FUNCTION_BLOCK INTERNAL FB_StringBuilderEx_Any_Tests EXTENDS TcUnit.FB_TestSuite
VAR_INPUT
END_VAR
VAR_OUTPUT
END_VAR
VAR
	stringBuilder	: FB_StringBuilder;
END_VAR

Test01_BOOL();
Test02_BYTE();
Test03_DATE();
Test04_DateAndTime();
Test05_DINT();
Test06_DWORD();
Test07_ENUM();
Test08_INT();
Test09_LINT();
Test10_LREAL();
Test11_LTIME();
Test12_LWORD();
Test13_REAL();
Test14_SINT();
Test15_STRING();
Test16_TIME();
Test17_TOD();
Test18_UDINT();
Test19_UINT();
Test20_ULINT();
Test21_USINT();
Test22_WORD();
Test23_WSTRING();
Test24_ANY_BIT_WORD();
Test25_ANY_BIT_BYTE();
Test26_ANY_BIT_DWORD();
Test27_ANY_BIT_LWORD();
Test28_ANY_REAL_REAL();
Test29_ANY_REAL_LREAL();

METHOD Test01_BOOL
VAR_INPUT
END_VAR

VAR_INST
	bTrue		: BOOL := TRUE;
	bFalse		: BOOL := FALSE;

END_VAR
IF TcUnit.TEST_ORDERED('Test01_BOOL') THEN
	AssertEquals_STRING(
		Actual := stringBuilder.Reset().AddAny(bTrue).Create(),
		Expected := 'TRUE',
		Message := 'Adding boolean failed');
		
	AssertEquals_STRING(
		Actual := stringBuilder.Reset().AddAny(bFalse).Create(),
		Expected := 'FALSE',
		Message := 'Adding boolean failed');
		
	TcUnit.TEST_FINISHED();
END_IF
END_METHOD

METHOD Test02_BYTE
VAR_INPUT
END_VAR
VAR
	byteVar	: BYTE := 17;
END_VAR
IF TEST_ORDERED('Test02_BYTE') THEN
	
	AssertEquals_STRING(
		Actual := stringBuilder.Reset().AddAny(byteVar).Create(),
		Expected := '17',
		Message := 'Adding BYTE failed.');
	TEST_FINISHED();
END_IF
END_METHOD

METHOD Test03_DATE
VAR
	someVar	: DATE := D#1970-01-01;
END_VAR
IF TEST_ORDERED('Test03_DATE') THEN
	AssertEquals_STRING(
		Actual := stringBuilder.Reset().AddAny(someVar).Create(),
		Expected := 'D#1970-01-01',
		Message := 'Adding DATE failed.');

	TEST_FINISHED();
END_IF
END_METHOD

METHOD Test04_DateAndTime
VAR
	someVar	: DATE_AND_TIME := DT#1970-1-1-0:0:1;
END_VAR
IF TEST_ORDERED('Test04_DateAndTime') THEN
	AssertEquals_STRING(
		Actual := stringBuilder.Reset().AddAny(someVar).Create(),
		Expected := 'DT#1970-01-01-00:00:01',
		Message := 'Adding DATE_AND_TIME failed.');

	TEST_FINISHED();
END_IF
END_METHOD

METHOD Test05_DINT
VAR
	someVar	: DINT := 15;
END_VAR
IF TEST_ORDERED('Test05_DINT') THEN
	AssertEquals_STRING(
		Actual := stringBuilder.Reset().AddAny(someVar).Create(),
		Expected := '15',
		Message := 'Adding DINT failed.');

	TEST_FINISHED();
END_IF
END_METHOD

METHOD Test06_DWORD
VAR
	someVar	: DWORD := 777;
END_VAR
IF TEST_ORDERED('Test06_DWORD') THEN
	AssertEquals_STRING(
		Actual := stringBuilder.Reset().AddAny(someVar).Create(),
		Expected := '777',
		Message := 'Adding DWORD failed.');

	TEST_FINISHED();
END_IF
END_METHOD

METHOD Test07_ENUM
VAR
	someVar	: E_AddAnyBitOptions := E_AddAnyBitOptions.HEXADECIMAL;
END_VAR
IF TEST_ORDERED('Test07_ENUM') THEN
	AssertEquals_STRING(
		Actual := stringBuilder.Reset().AddAny(someVar).Create(),
		Expected := '2',
		Message := 'Adding ENUM failed.');

	TEST_FINISHED();
END_IF
END_METHOD

METHOD Test08_INT
VAR
	someVar	: INT := 22;
END_VAR
IF TEST_ORDERED('Test08_INT') THEN
	AssertEquals_STRING(
		Actual := stringBuilder.Reset().AddAny(someVar).Create(),
		Expected := '22',
		Message := 'Adding INT failed.');

	TEST_FINISHED();
END_IF
END_METHOD

METHOD Test09_LINT
VAR
	someVar	: LINT := 6666;
END_VAR
IF TEST_ORDERED('Test09_LINT') THEN
	AssertEquals_STRING(
		Actual := stringBuilder.Reset().AddAny(someVar).Create(),
		Expected := '6666',
		Message := 'Adding LINT failed.');

	TEST_FINISHED();
END_IF
END_METHOD

METHOD Test10_LREAL
VAR
	someVar	: LREAL := 11.11;
END_VAR
IF TEST_ORDERED('Test10_LREAL') THEN
	AssertEquals_STRING(
		Actual := stringBuilder.Reset().AddAny(someVar).Create(),
		Expected := '11.11',
		Message := 'Adding LREAL failed.');

	TEST_FINISHED();
END_IF
END_METHOD

METHOD Test11_LTIME
VAR
	someVar	: LTIME := LTIME#100D2H30M40S500MS600US700NS;
END_VAR
IF TEST_ORDERED('Test11_LTIME') THEN
	AssertEquals_STRING(
		Actual := stringBuilder.Reset().AddAny(someVar).Create(),
		Expected := 'LTIME#100d2h30m40s500ms600us700ns',
		Message := 'Adding LTIME failed.');

	TEST_FINISHED();
END_IF
END_METHOD

METHOD Test12_LWORD
VAR
	someVar	: LWORD := 123456;
END_VAR
IF TEST_ORDERED('Test12_LWORD') THEN
	AssertEquals_STRING(
		Actual := stringBuilder.Reset().AddAny(someVar).Create(),
		Expected := '123456',
		Message := 'Adding LWORD failed.');

	TEST_FINISHED();
END_IF
END_METHOD

METHOD Test13_REAL
VAR
	someVar	: REAL := 12345.6789;
END_VAR
IF TEST_ORDERED('Test13_REAL') THEN
	AssertEquals_STRING(
		Actual := stringBuilder.Reset().AddAny(someVar).Create(),
		Expected := '12345.679',
		Message := 'Adding REAL failed.');

	TEST_FINISHED();
END_IF
END_METHOD

METHOD Test14_SINT
VAR
	someVar	: SINT := -34;
END_VAR
IF TEST_ORDERED('Test14_SINT') THEN
	AssertEquals_STRING(
		Actual := stringBuilder.Reset().AddAny(someVar).Create(),
		Expected := '-34',
		Message := 'Adding SINT failed.');

	TEST_FINISHED();
END_IF
END_METHOD

METHOD Test15_STRING
VAR
	someVar	: STRING := 'haha';
END_VAR
IF TEST_ORDERED('Test15_STRING') THEN
	AssertEquals_STRING(
		Actual := stringBuilder.Reset().AddAny(someVar).Create(),
		Expected := 'haha',
		Message := 'Adding STRING failed.');

	TEST_FINISHED();
END_IF
END_METHOD

METHOD Test16_TIME
VAR
	someVar	: TIME := T#15D10S;
END_VAR
IF TEST_ORDERED('Test16_TIME') THEN
	AssertEquals_STRING(
		Actual := stringBuilder.Reset().AddAny(someVar).Create(),
		Expected := 'T#15d10s',
		Message := 'Adding TIME failed.');

	TEST_FINISHED();
END_IF
END_METHOD

METHOD Test17_TOD
VAR
	someVar	: TOD := TOD#14:01:05.123;
END_VAR
IF TEST_ORDERED('Test17_TOD') THEN
	AssertEquals_STRING(
		Actual := stringBuilder.Reset().AddAny(someVar).Create(),
		Expected := 'TOD#14:01:05.123',
		Message := 'Adding TOD failed.');

	TEST_FINISHED();
END_IF
END_METHOD

METHOD Test18_UDINT
VAR
	someVar	: UDINT := 23452352;
END_VAR
IF TEST_ORDERED('Test18_UDINT') THEN
	AssertEquals_STRING(
		Actual := stringBuilder.Reset().AddAny(someVar).Create(),
		Expected := '23452352',
		Message := 'Adding UDINT failed.');

	TEST_FINISHED();
END_IF
END_METHOD

METHOD Test19_UINT
VAR
	someVar	: UINT := 12341;
END_VAR
IF TEST_ORDERED('Test19_UINT') THEN
	AssertEquals_STRING(
		Actual := stringBuilder.Reset().AddAny(someVar).Create(),
		Expected := '12341',
		Message := 'Adding UINT failed.');

	TEST_FINISHED();
END_IF
END_METHOD

METHOD Test20_ULINT
VAR
	someVar	: ULINT := 12345678;
END_VAR
IF TEST_ORDERED('Test20_ULINT') THEN
	AssertEquals_STRING(
		Actual := stringBuilder.Reset().AddAny(someVar).Create(),
		Expected := '12345678',
		Message := 'Adding ULINT failed.');

	TEST_FINISHED();
END_IF
END_METHOD

METHOD Test21_USINT
VAR
	someVar	: USINT := 123;
END_VAR
IF TEST_ORDERED('Test21_USINT') THEN
	AssertEquals_STRING(
		Actual := stringBuilder.Reset().AddAny(someVar).Create(),
		Expected := '123',
		Message := 'Adding USINT failed.');

	TEST_FINISHED();
END_IF
END_METHOD

METHOD Test22_WORD
VAR
	someVar	: WORD := 16#A;
END_VAR
IF TEST_ORDERED('Test22_WORD') THEN
	AssertEquals_STRING(
		Actual := stringBuilder.Reset().AddAny(someVar).Create(),
		Expected := '10',
		Message := 'Adding WORD failed.');

	TEST_FINISHED();
END_IF
END_METHOD

METHOD Test23_WSTRING
VAR
	someVar	: WSTRING := "test";
END_VAR
IF TEST_ORDERED('Test23_WSTRING') THEN
	AssertEquals_STRING(
		Actual := stringBuilder.Reset().AddAny(someVar).Create(),
		Expected := 'test',
		Message := 'Adding WSTRING failed.');

	TEST_FINISHED();
END_IF
END_METHOD

METHOD Test24_ANY_BIT_WORD
VAR_INPUT
END_VAR
VAR
	wordVar	: WORD := 16#AB;
	result	: Tc2_System.T_MaxString;
END_VAR
IF TcUnit.TEST_ORDERED('Test24_ANY_BIT_WORD') THEN
	
	// BINARY with notations
	result := stringBuilder.Reset().
		AddAnyBit(
			anyBit := wordVar, 
			option := E_AddAnyBitOptions.BINARY, 
			lowerCase := FALSE, 
			displayedDigitsCount := 16, 
			addNotation := TRUE)
		.Create();
		
	AssertEquals_STRING(
		Actual := result,
		Expected := '(BIN)0000000010101011',
		Message := 'Adding word as BINARY with addNotation = TRUE was incorrect');
		
	// BINARY without notations
	result := stringBuilder.Reset()
		.AddAnyBit(
			anyBit := wordVar, 
			option := E_AddAnyBitOptions.BINARY, 
			lowerCase := FALSE, 
			displayedDigitsCount := 16, 
			addNotation := FALSE)
		.Create();
		
	AssertEquals_STRING(
		Actual := result,
		Expected := '0000000010101011',
		Message := 'Adding word as BINARY with addNotation = FALSE was incorrect');
		
	// DECIMAL with notations
	result := stringBuilder.Reset()
		.AddAnyBit(
			anyBit := wordVar, 
			option := E_AddAnyBitOptions.DECIMAL, 
			lowerCase := FALSE, 
			displayedDigitsCount := 16, 
			addNotation := TRUE)
		.Create();
		
	AssertEquals_STRING(
		Actual := result,
		Expected := '(DEC)0000000000000171',
		Message := 'Adding word as DECIMAL with addNotation = TRUE was incorrect');
		
	// DECIMAL without notations
	result := stringBuilder.Reset()
		.AddAnyBit(
			anyBit := wordVar, 
			option := E_AddAnyBitOptions.DECIMAL, 
			lowerCase := FALSE, 
			displayedDigitsCount := 16, 
			addNotation := FALSE)
		.Create();
		
	AssertEquals_STRING(
		Actual := result,
		Expected := '0000000000000171',
		Message := 'Adding word as DECIMAL with addNotation = FALSE was incorrect');

	// HEXADECIMAL with notations
	result := stringBuilder.Reset()
		.AddAnyBit(
			anyBit := wordVar, 
			option := E_AddAnyBitOptions.HEXADECIMAL, 
			lowerCase := FALSE, 
			displayedDigitsCount := 16, 
			addNotation := TRUE)
		.Create();
		
	AssertEquals_STRING(
		Actual := result,
		Expected := '(HEX)00000000000000AB',
		Message := 'Adding word as HEXADECIMAL with addNotation = TRUE was incorrect');
		
	// HEXADECIMAL without notations
	result := stringBuilder.Reset()
		.AddAnyBit(
			anyBit := wordVar, 
			option := E_AddAnyBitOptions.HEXADECIMAL, 
			lowerCase := FALSE, 
			displayedDigitsCount := 16, 
			addNotation := FALSE)
		.Create();
		
	AssertEquals_STRING(
		Actual := result,
		Expected := '00000000000000AB',
		Message := 'Adding word as HEXADECIMAL with addNotation = FALSE was incorrect');
	
	// OCTAL with notations
	result := stringBuilder.Reset()
		.AddAnyBit(
			anyBit := wordVar, 
			option := E_AddAnyBitOptions.OCTAL, 
			lowerCase := FALSE, 
			displayedDigitsCount := 16, 
			addNotation := TRUE)
		.Create();
		
	AssertEquals_STRING(
		Actual := result,
		Expected := '(OCT)0000000000000253',
		Message := 'Adding word as OCTAL with addNotation = TRUE was incorrect');
		
	// OCTAL without notations
	result := stringBuilder.Reset()
		.AddAnyBit(
			anyBit := wordVar, 
			option := E_AddAnyBitOptions.OCTAL, 
			lowerCase := FALSE, 
			displayedDigitsCount := 16, 
			addNotation := FALSE)
		.Create();
		
	AssertEquals_STRING(
		Actual := result,
		Expected := '0000000000000253',
		Message := 'Adding word as OCTAL with addNotation = FALSE was incorrect');
		
	TcUnit.TEST_FINISHED();
END_IF
END_METHOD

METHOD Test25_ANY_BIT_BYTE
VAR_INPUT
END_VAR
VAR
	byteVar	: BYTE := 16#AB;
	result	: Tc2_System.T_MaxString;
END_VAR
IF TcUnit.TEST_ORDERED('Test25_ANY_BIT_BYTE') THEN
	
	// BINARY with notations
	result := stringBuilder.Reset().
		AddAnyBit(
			anyBit := byteVar, 
			option := E_AddAnyBitOptions.BINARY, 
			lowerCase := FALSE, 
			displayedDigitsCount := 8, 
			addNotation := TRUE)
		.Create();
		
	AssertEquals_STRING(
		Actual := result,
		Expected := '(BIN)10101011',
		Message := 'Adding byte as BINARY with addNotation = TRUE was incorrect');
		
	// BINARY without notations
	result := stringBuilder.Reset()
		.AddAnyBit(
			anyBit := byteVar, 
			option := E_AddAnyBitOptions.BINARY, 
			lowerCase := FALSE, 
			displayedDigitsCount := 8, 
			addNotation := FALSE)
		.Create();
		
	AssertEquals_STRING(
		Actual := result,
		Expected := '10101011',
		Message := 'Adding byte as BINARY with addNotation = FALSE was incorrect');
		
	// DECIMAL with notations
	result := stringBuilder.Reset()
		.AddAnyBit(
			anyBit := byteVar, 
			option := E_AddAnyBitOptions.DECIMAL, 
			lowerCase := FALSE, 
			displayedDigitsCount := 8, 
			addNotation := TRUE)
		.Create();
		
	AssertEquals_STRING(
		Actual := result,
		Expected := '(DEC)00000171',
		Message := 'Adding byte as DECIMAL with addNotation = TRUE was incorrect');
		
	// DECIMAL without notations
	result := stringBuilder.Reset()
		.AddAnyBit(
			anyBit := byteVar, 
			option := E_AddAnyBitOptions.DECIMAL, 
			lowerCase := FALSE, 
			displayedDigitsCount := 8, 
			addNotation := FALSE)
		.Create();
		
	AssertEquals_STRING(
		Actual := result,
		Expected := '00000171',
		Message := 'Adding byte as DECIMAL with addNotation = FALSE was incorrect');

	// HEXADECIMAL with notations
	result := stringBuilder.Reset()
		.AddAnyBit(
			anyBit := byteVar, 
			option := E_AddAnyBitOptions.HEXADECIMAL, 
			lowerCase := FALSE, 
			displayedDigitsCount := 8, 
			addNotation := TRUE)
		.Create();
		
	AssertEquals_STRING(
		Actual := result,
		Expected := '(HEX)000000AB',
		Message := 'Adding byte as HEXADECIMAL with addNotation = TRUE was incorrect');
		
	// HEXADECIMAL without notations
	result := stringBuilder.Reset()
		.AddAnyBit(
			anyBit := byteVar, 
			option := E_AddAnyBitOptions.HEXADECIMAL, 
			lowerCase := FALSE, 
			displayedDigitsCount := 8, 
			addNotation := FALSE)
		.Create();
		
	AssertEquals_STRING(
		Actual := result,
		Expected := '000000AB',
		Message := 'Adding byte as HEXADECIMAL with addNotation = FALSE was incorrect');
	
	// OCTAL with notations
	result := stringBuilder.Reset()
		.AddAnyBit(
			anyBit := byteVar, 
			option := E_AddAnyBitOptions.OCTAL, 
			lowerCase := FALSE, 
			displayedDigitsCount := 8, 
			addNotation := TRUE)
		.Create();
		
	AssertEquals_STRING(
		Actual := result,
		Expected := '(OCT)00000253',
		Message := 'Adding byte as OCTAL with addNotation = TRUE was incorrect');
		
	// OCTAL without notations
	result := stringBuilder.Reset()
		.AddAnyBit(
			anyBit := byteVar, 
			option := E_AddAnyBitOptions.OCTAL, 
			lowerCase := FALSE, 
			displayedDigitsCount := 8, 
			addNotation := FALSE)
		.Create();
		
	AssertEquals_STRING(
		Actual := result,
		Expected := '00000253',
		Message := 'Adding byte as OCTAL with addNotation = FALSE was incorrect');
		
	TcUnit.TEST_FINISHED();
END_IF
END_METHOD

METHOD Test26_ANY_BIT_DWORD
VAR
	dwordVar	: DWORD := 16#AB;
	result	: Tc2_System.T_MaxString;
END_VAR
IF TcUnit.TEST_ORDERED('Test26_ANY_BIT_DWORD') THEN
	
	// BINARY with notations
	result := stringBuilder.Reset().
		AddAnyBit(
			anyBit := dwordVar, 
			option := E_AddAnyBitOptions.BINARY, 
			lowerCase := FALSE, 
			displayedDigitsCount := 32, 
			addNotation := TRUE)
		.Create();
		
	AssertEquals_STRING(
		Actual := result,
		Expected := '(BIN)00000000000000000000000010101011',
		Message := 'Adding dword as BINARY with addNotation = TRUE was incorrect');
		
	// BINARY without notations
	result := stringBuilder.Reset()
		.AddAnyBit(
			anyBit := dwordVar, 
			option := E_AddAnyBitOptions.BINARY, 
			lowerCase := FALSE, 
			displayedDigitsCount := 32, 
			addNotation := FALSE)
		.Create();
		
	AssertEquals_STRING(
		Actual := result,
		Expected := '00000000000000000000000010101011',
		Message := 'Adding dword as BINARY with addNotation = FALSE was incorrect');
		
	// DECIMAL with notations
	result := stringBuilder.Reset()
		.AddAnyBit(
			anyBit := dwordVar, 
			option := E_AddAnyBitOptions.DECIMAL, 
			lowerCase := FALSE, 
			displayedDigitsCount := 32, 
			addNotation := TRUE)
		.Create();
		
	AssertEquals_STRING(
		Actual := result,
		Expected := '(DEC)00000000000000000000000000000171',
		Message := 'Adding dword as DECIMAL with addNotation = TRUE was incorrect');
		
	// DECIMAL without notations
	result := stringBuilder.Reset()
		.AddAnyBit(
			anyBit := dwordVar, 
			option := E_AddAnyBitOptions.DECIMAL, 
			lowerCase := FALSE, 
			displayedDigitsCount := 32, 
			addNotation := FALSE)
		.Create();
		
	AssertEquals_STRING(
		Actual := result,
		Expected := '00000000000000000000000000000171',
		Message := 'Adding dword as DECIMAL with addNotation = FALSE was incorrect');

	// HEXADECIMAL with notations
	result := stringBuilder.Reset()
		.AddAnyBit(
			anyBit := dwordVar, 
			option := E_AddAnyBitOptions.HEXADECIMAL, 
			lowerCase := FALSE, 
			displayedDigitsCount := 32, 
			addNotation := TRUE)
		.Create();
		
	AssertEquals_STRING(
		Actual := result,
		Expected := '(HEX)000000000000000000000000000000AB',
		Message := 'Adding dword as HEXADECIMAL with addNotation = TRUE was incorrect');
		
	// HEXADECIMAL without notations
	result := stringBuilder.Reset()
		.AddAnyBit(
			anyBit := dwordVar, 
			option := E_AddAnyBitOptions.HEXADECIMAL, 
			lowerCase := FALSE, 
			displayedDigitsCount := 32, 
			addNotation := FALSE)
		.Create();
		
	AssertEquals_STRING(
		Actual := result,
		Expected := '000000000000000000000000000000AB',
		Message := 'Adding dword as HEXADECIMAL with addNotation = FALSE was incorrect');
	
	// OCTAL with notations
	result := stringBuilder.Reset()
		.AddAnyBit(
			anyBit := dwordVar, 
			option := E_AddAnyBitOptions.OCTAL, 
			lowerCase := FALSE, 
			displayedDigitsCount := 32, 
			addNotation := TRUE)
		.Create();
		
	AssertEquals_STRING(
		Actual := result,
		Expected := '(OCT)00000000000000000000000000000253',
		Message := 'Adding dword as OCTAL with addNotation = TRUE was incorrect');
		
	// OCTAL without notations
	result := stringBuilder.Reset()
		.AddAnyBit(
			anyBit := dwordVar, 
			option := E_AddAnyBitOptions.OCTAL, 
			lowerCase := FALSE, 
			displayedDigitsCount := 32, 
			addNotation := FALSE)
		.Create();
		
	AssertEquals_STRING(
		Actual := result,
		Expected := '00000000000000000000000000000253',
		Message := 'Adding dword as OCTAL with addNotation = FALSE was incorrect');
		
	TcUnit.TEST_FINISHED();
END_IF
END_METHOD

METHOD Test27_ANY_BIT_LWORD
VAR
	lwordVar	: LWORD := 16#AB;
	result	: Tc2_System.T_MaxString;
END_VAR
IF TcUnit.TEST_ORDERED('Test27_ANY_BIT_LWORD') THEN
	
	// BINARY with notations
	result := stringBuilder.Reset().
		AddAnyBit(
			anyBit := lwordVar, 
			option := E_AddAnyBitOptions.BINARY, 
			lowerCase := FALSE, 
			displayedDigitsCount := 64, 
			addNotation := TRUE)
		.Create();
		
	AssertEquals_STRING(
		Actual := result,
		Expected := '(BIN)0000000000000000000000000000000000000000000000000000000010101011',
		Message := 'Adding lword as BINARY with addNotation = TRUE was incorrect');
		
	// BINARY without notations
	result := stringBuilder.Reset()
		.AddAnyBit(
			anyBit := lwordVar, 
			option := E_AddAnyBitOptions.BINARY, 
			lowerCase := FALSE, 
			displayedDigitsCount := 64, 
			addNotation := FALSE)
		.Create();
		
	AssertEquals_STRING(
		Actual := result,
		Expected := '0000000000000000000000000000000000000000000000000000000010101011',
		Message := 'Adding lword as BINARY with addNotation = FALSE was incorrect');
		
	// DECIMAL with notations
	result := stringBuilder.Reset()
		.AddAnyBit(
			anyBit := lwordVar, 
			option := E_AddAnyBitOptions.DECIMAL, 
			lowerCase := FALSE, 
			displayedDigitsCount := 64, 
			addNotation := TRUE)
		.Create();
		
	AssertEquals_STRING(
		Actual := result,
		Expected := '(DEC)0000000000000000000000000000000000000000000000000000000000000171',
		Message := 'Adding lword as DECIMAL with addNotation = TRUE was incorrect');
		
	// DECIMAL without notations
	result := stringBuilder.Reset()
		.AddAnyBit(
			anyBit := lwordVar, 
			option := E_AddAnyBitOptions.DECIMAL, 
			lowerCase := FALSE, 
			displayedDigitsCount := 64, 
			addNotation := FALSE)
		.Create();
		
	AssertEquals_STRING(
		Actual := result,
		Expected := '0000000000000000000000000000000000000000000000000000000000000171',
		Message := 'Adding lword as DECIMAL with addNotation = FALSE was incorrect');

	// HEXADECIMAL with notations
	result := stringBuilder.Reset()
		.AddAnyBit(
			anyBit := lwordVar, 
			option := E_AddAnyBitOptions.HEXADECIMAL, 
			lowerCase := FALSE, 
			displayedDigitsCount := 64, 
			addNotation := TRUE)
		.Create();
		
	AssertEquals_STRING(
		Actual := result,
		Expected := '(HEX)00000000000000000000000000000000000000000000000000000000000000AB',
		Message := 'Adding lword as HEXADECIMAL with addNotation = TRUE was incorrect');
		
	// HEXADECIMAL without notations
	result := stringBuilder.Reset()
		.AddAnyBit(
			anyBit := lwordVar, 
			option := E_AddAnyBitOptions.HEXADECIMAL, 
			lowerCase := FALSE, 
			displayedDigitsCount := 64, 
			addNotation := FALSE)
		.Create();
		
	AssertEquals_STRING(
		Actual := result,
		Expected := '00000000000000000000000000000000000000000000000000000000000000AB',
		Message := 'Adding lword as HEXADECIMAL with addNotation = FALSE was incorrect');
	
	// OCTAL with notations
	result := stringBuilder.Reset()
		.AddAnyBit(
			anyBit := lwordVar, 
			option := E_AddAnyBitOptions.OCTAL, 
			lowerCase := FALSE, 
			displayedDigitsCount := 64, 
			addNotation := TRUE)
		.Create();
		
	AssertEquals_STRING(
		Actual := result,
		Expected := '(OCT)0000000000000000000000000000000000000000000000000000000000000253',
		Message := 'Adding lword as OCTAL with addNotation = TRUE was incorrect');
		
	// OCTAL without notations
	result := stringBuilder.Reset()
		.AddAnyBit(
			anyBit := lwordVar, 
			option := E_AddAnyBitOptions.OCTAL, 
			lowerCase := FALSE, 
			displayedDigitsCount := 64, 
			addNotation := FALSE)
		.Create();
		
	AssertEquals_STRING(
		Actual := result,
		Expected := '0000000000000000000000000000000000000000000000000000000000000253',
		Message := 'Adding lword as OCTAL with addNotation = FALSE was incorrect');
		
	TcUnit.TEST_FINISHED();
END_IF
END_METHOD

METHOD Test28_ANY_REAL_REAL
VAR
	realVar	: REAL := 12345.123888;
	result	: Tc2_System.T_MaxString;
END_VAR
IF TcUnit.TEST_ORDERED('Test28_ANY_REAL_REAL') THEN
	result := stringBuilder.Reset().
		AddAnyReal(
			anyReal := realVar,
			precision := 2,
			round := FALSE)
		.Create();	

	AssertEquals_STRING(
		Actual := result,
		Expected := '12345.12',
		Message := 'Adding REAL with round = FALSE failed.');
		
	result := stringBuilder.Reset().
		AddAnyReal(
			anyReal := realVar,
			precision := 3,
			round := TRUE)
		.Create();	

	AssertEquals_STRING(
		Actual := result,
		Expected := '12345.124',
		Message := 'Adding REAL with round = TRUE failed.');
		
	TcUnit.TEST_FINISHED();
END_IF
END_METHOD

METHOD Test29_ANY_REAL_LREAL
VAR
	lrealVar	: LREAL := 12345.12345678;
	result	: Tc2_System.T_MaxString;
END_VAR
IF TcUnit.TEST_ORDERED('Test29_ANY_REAL_LREAL') THEN
	result := stringBuilder.Reset().
		AddAnyReal(
			anyReal := lrealVar,
			precision := 5,
			round := FALSE)
		.Create();	

	AssertEquals_STRING(
		Actual := result,
		Expected := '12345.12345',
		Message := 'Adding LREAL with round = FALSE failed.');
		
	result := stringBuilder.Reset().
		AddAnyReal(
			anyReal := lrealVar,
			precision := 7,
			round := TRUE)
		.Create();	

	AssertEquals_STRING(
		Actual := result,
		Expected := '12345.1234568',
		Message := 'Adding LREAL with round = TRUE failed.');
		
	TcUnit.TEST_FINISHED();
END_IF
END_METHOD

END_FUNCTION_BLOCK

(* stored: Version 1.1.0.1, ProductVersion 3.1.4024.14
   POU FB_StringBuilderEx_Any_Tests: Id {993fbc3e-5c9d-0f17-0385-4fce2f3aa1dd}, SpecialFunc None
   Method Test01_BOOL: Id {cfb9a40b-eb82-0aeb-29ca-569dd72e79c7}
   Method Test02_BYTE: Id {c4fd4cb4-7ad4-0c82-28ce-eca0288b2bd4}
   Method Test03_DATE: Id {2e1f0d36-48a6-0114-01e4-b61e830c0de7}
   Method Test04_DateAndTime: Id {43674567-cbf3-0b60-3a1a-25c0832a193a}
   Method Test05_DINT: Id {d74a7aab-7f5a-0848-0fd8-3c29d1e1cf1d}
   Method Test06_DWORD: Id {8f64b908-2c4e-05d5-1577-c9f32c694f35}
   Method Test07_ENUM: Id {71268857-77ee-0509-1941-f38bd3e4031a}
   Method Test08_INT: Id {50412636-13a0-03e7-292c-fcb255f8bd55}
   Method Test09_LINT: Id {8005f92e-a205-0e43-38d5-826ab2a0292f}
   Method Test10_LREAL: Id {9113eedd-ee6c-0191-2fe7-457e71b3657e}
   Method Test11_LTIME: Id {fc4e2ed8-904a-075b-1438-0244b9d03c7f}
   Method Test12_LWORD: Id {b67d9c3d-52b4-0b6b-35cf-913ba29a6594}
   Method Test13_REAL: Id {2816e998-89c0-096b-3a74-9a11ab704eb8}
   Method Test14_SINT: Id {6c7665bf-0153-0ce1-0e35-d654cb2ce2aa}
   Method Test15_STRING: Id {94253549-fafe-0f80-09c6-89ebc1d88293}
   Method Test16_TIME: Id {2160ef82-12b9-0d94-27e9-4339ba76733c}
   Method Test17_TOD: Id {d7841bc8-20ff-0ac3-2e6d-e7ec37f51186}
   Method Test18_UDINT: Id {bd53d0e6-72cd-0c1c-1e1f-e2cba32aa961}
   Method Test19_UINT: Id {fe13564c-b104-0e32-105a-b836699707c7}
   Method Test20_ULINT: Id {bd8cb3b1-9a8b-0c9a-2994-527d8693f902}
   Method Test21_USINT: Id {22dcfb33-d0bc-0d5f-3114-b0b2104acc31}
   Method Test22_WORD: Id {ab55a167-5334-0617-2b2d-8531f2f2e240}
   Method Test23_WSTRING: Id {7b808dee-1ef7-0617-2d8c-b16a5c3b233b}
   Method Test24_ANY_BIT_WORD: Id {cb289a5e-b78c-01b6-05a8-fb68091cd4fb}
   Method Test25_ANY_BIT_BYTE: Id {3e550e7b-2522-0e59-252d-d1f17213e7d2}
   Method Test26_ANY_BIT_DWORD: Id {d34ecae9-fdb6-0c8a-1e30-9d1313ab862c}
   Method Test27_ANY_BIT_LWORD: Id {f929254d-fa61-062f-0af3-37cbe0ae0a1d}
   Method Test28_ANY_REAL_REAL: Id {6d237f3d-660f-087b-1049-692edac18b97}
   Method Test29_ANY_REAL_LREAL: Id {7049dc39-845e-069a-24dd-c1ad1129622a} *)
